FUNCTION_BLOCK ImagesToVideo
VAR_INPUT
	ImageExportPath	: STRING(255);
	VideoFilePath	: STRING(255);
	JSONAttribute	: STRING(255);
	
END_VAR
VAR_OUTPUT
	bBusy	: BOOL;
	bError	: BOOL;
	nErrID	: UDINT;
END_VAR
VAR
	Listener	: FB_ListenerBase2;
	EventFilter	: FB_TcEventFilter;
	hr			: HRESULT; 
END_VAR

//Listener.Execute();

//Filter out events using JSON attribute
//IF EventFilter.Clear().JsonAttribute = JSONAttribute THEN
//	hr := Listener.Subscribe2(EventFilter);
//END_IF

//Call

END_FUNCTION_BLOCK

(* stored: Version 1.1.0.1, ProductVersion 3.1.4024.10
   POU ImagesToVideo: Id {4ed94054-832b-00ce-312f-2065dce12fa2}, SpecialFunc None *)
